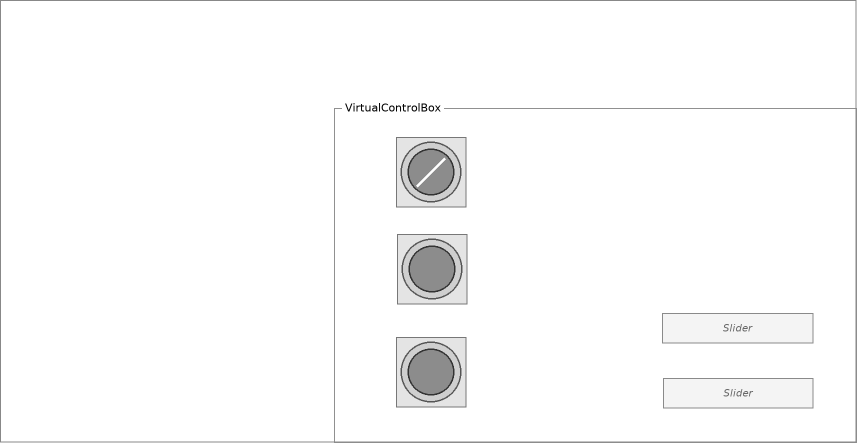
VISUALIZATION VirtualControlBox  // 857x443
    GroupBox (334,100 523x343), "VirtualControlBox"
        RotarySwitch (62,37 70x70), behaviour: TOGGLE, style: Switch-RotarySwitch-Gray
        PushSwitchLed (63,134 70x70), behaviour: TOGGLE, style: Switch-PushSwitchLed-Gray
        PushSwitchLed (62,237 70x70), behaviour: TOGGLE, style: Switch-PushSwitchLed-Gray
        Slider (329,278 150x30), scale 0..100
        Slider (328,213 151x30), scale 0..100
END_VISUALIZATION

(* stored: Version 1.1.0.1, ProductVersion 3.1.4024.12
   Visu VirtualControlBox: Id {c919442a-26ea-45f3-adf0-884bbcdf1b35} *)
